TYPE eMotorState :
(Idle,Accelerating,Running,Decelerating,Error)
END_TYPE

(* stored: Version 1.1.0.1, ProductVersion 3.1.4024.12
   DUT eMotorState: Id {c3d4e5f6-a7b8-4c9d-0e1f-2a3b4c5d6e7f} *)
